// TwinCAT 3 PLC project Untitled1
// ProgramVersion: 3.1.4024.0
// libraries:
//   Tc2_Standard, * (Beckhoff Automation GmbH)
//   Tc2_System, * (Beckhoff Automation GmbH)
//   Tc3_Module, * (Beckhoff Automation GmbH)
// project tree:
//   / PlcTask.TcTTO
//   POUs/ MAIN.TcPOU
// real-time tasks:
//   TASK PlcTask: cycle T#10ms, priority 20, ADS port 350
// I/O:
//   DEVICE Device 1 (Beckhoff CCAT)
//   DEVICE Device 2 (EtherCAT), AmsNetId 5.116.114.25.3.1
//     Term 1 (EK1200) [EK1200-5000 EtherCAT Power supply (2A E-Bus)]
//       Term 2 (EL2911) [EL2911, Potential supply terminal (10 A) with 4 Ch. Safety Inputs, TwinSAFE]
//         modules: Module 2 (FSOUT), Module 3 (DEVICEIO), Module 4 (FSLOGIC)
//       Term 3 (EK1110) [EK1110 EtherCAT extension]
//     Box 4 (MBM-EC-S4-MLI-3B) [MBM-EC-S4-MLI-3B (EtherCAT)]
//       modules: Module 1 (FSoE 8 Bytes), Module 2 (MBM DIAGNOSE EXTENDED), Module 3 (MGB2-L1-MLI-U-Y0000-BJ-136776 Diagnose Basic), Module 4 (MSM-1-P-CA-PPP-SW-ID-9000003), Module 5 (MSM-1-P-CA-B000W0-I8-168644 Diagnose Basic)
// variable links:
//   Device 2 (EtherCAT) <-> Device 2 (EtherCAT)/Box 4 (MBM-EC-S4-MLI-3B)
//     Term 1 (EK1200)/Term 2 (EL2911)/ConnectionOutputs/Message_7 RxPDO <-> Module 1 (FSoE 8 Bytes)/Inputs/FSOE
//   Device 2 (EtherCAT) <-> Device 2 (EtherCAT)/Term 1 (EK1200)/Term 2 (EL2911)
//     Box 4 (MBM-EC-S4-MLI-3B)/Module 1 (FSoE 8 Bytes)/Outputs/FSOE <-> ConnectionInputs/Message_7 TxPDO
//     Box 4 (MBM-EC-S4-MLI-3B)/Module 4 (MSM-1-P-CA-PPP-SW-ID-9000003)/Inputs/Input Byte 1 @bit 1 <-> StandardOutputs/Standard In Var 4
//     Box 4 (MBM-EC-S4-MLI-3B)/Module 4 (MSM-1-P-CA-PPP-SW-ID-9000003)/Inputs/Input Byte 1 <-> StandardOutputs/Standard In Var 5
//   Untitled1/Untitled1 Instance <-> Device 2 (EtherCAT)/Box 4 (MBM-EC-S4-MLI-3B)
//     PlcTask Outputs/MAIN.bAlwaysTrue <-> Module 3 (MGB2-L1-MLI-U-Y0000-BJ-136776 Diagnose Basic)/Outputs/Output Byte 1
//   Untitled1/Untitled1 Instance <-> Device 2 (EtherCAT)/Term 1 (EK1200)/Term 2 (EL2911)
//     PlcTask Outputs/MAIN.bErrAck <-> StandardOutputs/Standard In Var 1
//     PlcTask Outputs/MAIN.bRun <-> StandardOutputs/Standard In Var 2

CONFIGURATION Untitled1
    RESOURCE PLC ON TwinCAT3
        TASK PlcTask(INTERVAL := T#10ms, PRIORITY := 20);
        PROGRAM MAIN WITH PlcTask : MAIN;
    END_RESOURCE
END_CONFIGURATION

// ---- POUs/MAIN.TcPOU
PROGRAM MAIN
VAR
	
bAlwaysTrue  	AT%Q* 	: BOOL := TRUE;
bRun 		 	AT%Q* 	: BOOL;
bErrAck 		AT%Q*	: BOOL;

END_VAR

END_PROGRAM
